INTERFACE I_OutfeedModule

PROPERTY CfgOutfeed : REFERENCE TO ST_OutfeedConfig
GET
END_GET
END_PROPERTY

PROPERTY CmdOutfeed : REFERENCE TO ST_OutfeedCommand
GET
END_GET
END_PROPERTY

PROPERTY RcpOutfeed : REFERENCE TO ST_OutfeedRecipe
GET
END_GET
END_PROPERTY

PROPERTY StsOutfeed : REFERENCE TO ST_OutfeedStatus
GET
END_GET
END_PROPERTY

END_INTERFACE

(* stored: Version 1.1.0.1, ProductVersion 3.1.4024.12
   Itf I_OutfeedModule: Id {a270bc10-979d-4974-8beb-5485070ed871}
   Property CfgOutfeed: Id {b1204b23-659f-4873-90b0-0f83aa3678a2}
   Get Get: Id {51bcbe5f-92c0-44af-8a7c-1176a0fa0464}
   Property CmdOutfeed: Id {8176e77e-a962-4e76-96b9-57421a7e3c5e}
   Get Get: Id {6f786f40-8258-46c0-9440-50f278be1c9d}
   Property RcpOutfeed: Id {962c6e7c-a0fa-4160-80f6-85b4dcb6280c}
   Get Get: Id {2c772b01-7075-48a4-8033-c6faa9ea1c0d}
   Property StsOutfeed: Id {15a20845-7409-45b1-b7fc-6ac5eeace1ac}
   Get Get: Id {2fc23270-b8b3-42f0-b817-b56f91c808dd} *)
